{attribute 'GeneratedUsingTerminal: EL1512-0000-0017'}
{attribute addProperty BoxType "EL1512-0000-0017"}
{attribute addProperty Id "ControlAT %Q*Control_0B2F8B702Set_counter_valueAT %Q*UDINT4"}
{attribute addProperty CRC "1426831071"}
{attribute addProperty Size "6"}
TYPE CNT_Outputs_Channel_550BB6DF EXTENDS OutputBase_10CEE7DE :
STRUCT
	{attribute addProperty Name "Control"}
	Control AT %Q* : Control_0B2F8B70;
	{attribute addProperty Name "Set_counter_value"}
	Set_counter_value AT %Q* : UDINT;
END_STRUCT
END_TYPE

(* stored: Version 1.2.0.0, ProductVersion 3.1.4024.9
   DUT CNT_Outputs_Channel_550BB6DF: Id {298ba623-717d-4b3a-aaeb-50e56f6b03e7} *)
